RoboDK station: Enrega_Final.rdk

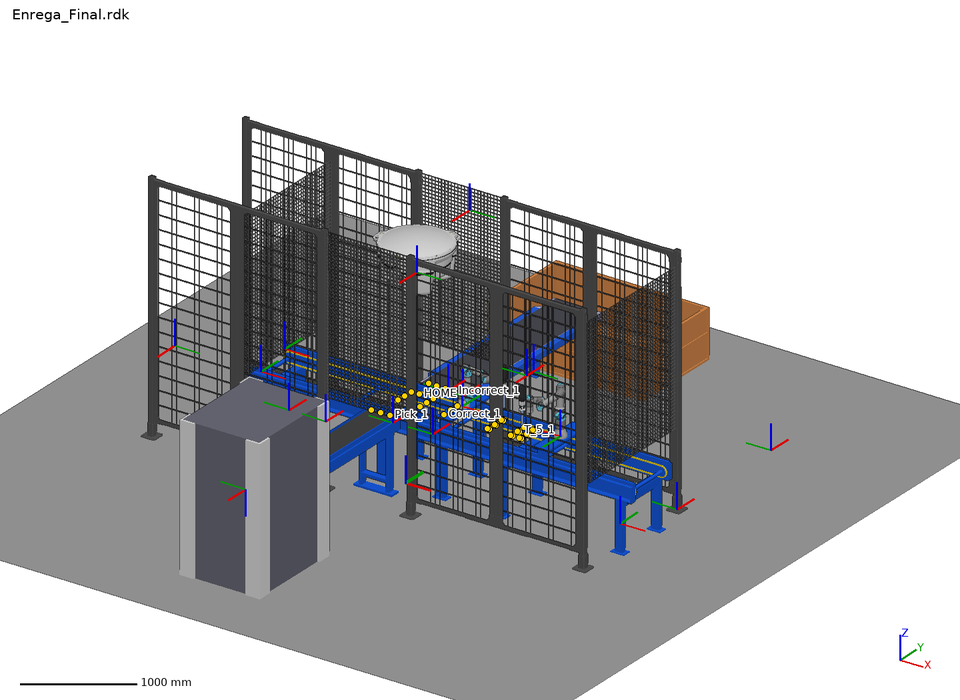
[picture v0: the station drawn from its stored meshes, robots at their saved joint values, targets as dots, program paths as lines]
Station Enrega_Final2 (saved by RoboDK 5.9.4). Poses are relative to the parent item; angles as X-Y-Z fixed-axis rotations.
Station parameters (name, value as stored): conv_pos, 0, groups_created, 0, stop, 0, group_counter_incorrectos, 0, conv_pos_exit, 0, groups_to_process, 0, serigrafia, 0, serigrafia1, 0, cinta_salida, 0, cinta_entrada, 0, salida_group_id, 0, salida_groups_on_belt, 0, salida_first_group_id, 0, main_conv_pos, 0, main_group_id, 0, main_groups_on_belt, 0, main_first_group_id, 0, cinta_central, 0, correct_group_id, 0, correct_groups_on_belt, 0, correct_first_group_id, 0, led_salida, 1, salir, 0
  - frame World at (0, 0, 0) mm
    - object Floor at (0, 0, 0) mm, size 7200 x 7200 x 0 mm, geometry from Floor.sld
    - frame MainConveyor Base at (-1580, 450, 650) mm
      - robot MainConveyor: 1 axes
          modified DH rows (alpha deg, a mm, theta deg, d mm): 0, 0, 0, 0 linear
          base shift (0, 0, 0) mm, rotated rx 0 ry 90 rz 0 deg
          joint limits [-200000] to [200000]; home [0]; saved at [0]
        - frame MainConveyorRef at (-800, -492, 0) mm, rotated rx 0 ry 0 rz -90 deg
      - frame MainConveyorRef_Init at (90, -480, 0) mm
    - frame UR3eBase1 at (1470, 200, 770) mm, rotated rx 0 ry 0 rz 180 deg
      - robot UR3e_1 (model UR3e): 6 axes, payload 3 kg, reach 500 mm, repeatability 0.03 mm, weight 11 kg
          modified DH rows (alpha deg, a mm, theta deg, d mm): 0, 0, 0, 151.9; 90, 0, 180, 0; 0, 243.55, 0, 0; 0, 213.2, 0, 131.05; -90, 0, 0, 85.35; 90, 0, 180, 92.1
          joint limits [-360, -360, -360, -360, -360, -360] to [360, 360, 360, 360, 360, 360]; home [0, -90, -90, 0, 90, 0]; saved at [38.708, -87.691, -123.564, -58.745, 90, 38.708]
        - tool Laser1, TCP at (0, -75, 221.24) mm, rotated rx 0 ry 0 rz 90 deg, size 63 x 128.2 x 432.2 mm
      - target T_5_1 (Cartesian target) at (453.12, -41.05, -88.71) mm, rotated rx -180 ry 0 rz -180 deg; joints [13.959, -117.749, -104.305, -47.946, 90, 13.959] of UR3e_1
      - target T_5_2 (Cartesian target) at (453.12, -31.05, -88.71) mm, rotated rx -180 ry 0 rz -180 deg; joints [15.513, -117.567, -104.617, -47.816, 90, 15.513] of UR3e_1
      - target T_5_3 (Cartesian target) at (453.12, -21.05, -88.71) mm, rotated rx -180 ry 0 rz -180 deg; joints [17.059, -117.435, -104.843, -47.722, 90, 17.059] of UR3e_1
      - target T_5_4 (Cartesian target) at (443.12, -21.05, -88.71) mm, rotated rx -180 ry 0 rz -180 deg; joints [17.546, -115.52, -108.09, -46.39, 90, 17.546] of UR3e_1
      - target T_5_5 (Cartesian target) at (463.12, -21.05, -88.71) mm, rotated rx -180 ry 0 rz -180 deg; joints [16.599, -119.355, -101.528, -49.117, 90, 16.599] of UR3e_1
      - target T_6_1 (Cartesian target) at (453.12, -141.05, -88.71) mm, rotated rx -180 ry 0 rz -180 deg; joints [-1.508, -122.242, -96.445, -51.314, 90, -1.508] of UR3e_1
      - target T_6_2 (Cartesian target) at (453.12, -131.05, -88.71) mm, rotated rx -180 ry 0 rz -180 deg; joints [0, -121.581, -97.617, -50.801, 90, 0] of UR3e_1
      - target T_6_3 (Cartesian target) at (453.12, -121.05, -88.71) mm, rotated rx -180 ry 0 rz -180 deg; joints [1.522, -120.967, -98.704, -50.329, 90, 1.522] of UR3e_1
      - target T_6_4 (Cartesian target) at (443.12, -121.05, -88.71) mm, rotated rx -180 ry 0 rz -180 deg; joints [1.564, -119.128, -101.923, -48.949, 90, 1.564] of UR3e_1
      - target T_6_5 (Cartesian target) at (463.12, -121.05, -88.71) mm, rotated rx -180 ry 0 rz -180 deg; joints [1.482, -122.826, -95.401, -51.773, 90, 1.482] of UR3e_1
      - target T_7_1 (Cartesian target) at (358.12, -136.05, -88.71) mm, rotated rx -180 ry 0 rz -180 deg; joints [-1.008, -104.831, -124.911, -40.258, 90, -1.008] of UR3e_1
      - target T_7_2 (Cartesian target) at (358.12, -126.05, -88.71) mm, rotated rx -180 ry 0 rz -180 deg; joints [1.016, -103.97, -126.152, -39.878, 90, 1.016] of UR3e_1
      - target T_7_3 (Cartesian target) at (358.12, -116.05, -88.71) mm, rotated rx -180 ry 0 rz -180 deg; joints [3.071, -103.155, -127.308, -39.536, 90, 3.071] of UR3e_1
      - target T_7_4 (Cartesian target) at (348.12, -116.05, -88.71) mm, rotated rx -180 ry 0 rz -180 deg; joints [3.186, -101.205, -130.002, -38.792, 90, 3.186] of UR3e_1
      - target T_7_5 (Cartesian target) at (368.12, -116.05, -88.71) mm, rotated rx -180 ry 0 rz -180 deg; joints [2.964, -105.064, -124.571, -40.364, 90, 2.964] of UR3e_1
      - target T_8_1 (Cartesian target) at (358.12, -41.05, -88.71) mm, rotated rx -180 ry 0 rz -180 deg; joints [19.014, -98.871, -133.084, -38.044, 90, 19.014] of UR3e_1
      - target T_8_2 (Cartesian target) at (358.12, -31.05, -88.71) mm, rotated rx -180 ry 0 rz -180 deg; joints [21.136, -98.589, -133.447, -37.965, 90, 21.136] of UR3e_1
      - target T_8_3 (Cartesian target) at (358.12, -21.05, -88.71) mm, rotated rx -180 ry 0 rz -180 deg; joints [23.239, -98.383, -133.709, -37.908, 90, 23.239] of UR3e_1
      - target T_8_4 (Cartesian target) at (348.12, -21.05, -88.71) mm, rotated rx -180 ry 0 rz -180 deg; joints [24.174, -96.082, -136.551, -37.367, 90, 24.174] of UR3e_1
      - target T_8_5 (Cartesian target) at (368.12, -21.05, -88.71) mm, rotated rx -180 ry 0 rz -180 deg; joints [22.376, -100.585, -130.837, -38.578, 90, 22.376] of UR3e_1
      - target T_9_1 (Cartesian target) at (358.12, 58.95, -88.71) mm, rotated rx -180 ry 0 rz -180 deg; joints [38.708, -99.562, -132.189, -38.249, 90, 38.708] of UR3e_1
      - target T_9_2 (Cartesian target) at (358.12, 68.95, -88.71) mm, rotated rx -180 ry 0 rz -180 deg; joints [40.414, -100.046, -131.554, -38.401, 90, 40.414] of UR3e_1
      - target T_9_3 (Cartesian target) at (358.12, 78.95, -88.71) mm, rotated rx -180 ry 0 rz -180 deg; joints [42.06, -100.595, -130.823, -38.581, 90, 42.06] of UR3e_1
      - target T_9_4 (Cartesian target) at (348.12, 78.95, -88.71) mm, rotated rx -180 ry 0 rz -180 deg; joints [43.571, -98.473, -133.594, -37.933, 90, 43.571] of UR3e_1
      - target T_9_5 (Cartesian target) at (368.12, 78.95, -88.71) mm, rotated rx -180 ry 0 rz -180 deg; joints [40.65, -102.65, -128.016, -39.334, 90, 40.65] of UR3e_1
    - frame UR3eBase2 at (450, 200, 770) mm
      - robot UR3e_2 (model UR3e): 6 axes, payload 3 kg, reach 500 mm, repeatability 0.03 mm, weight 11 kg
          modified DH rows (alpha deg, a mm, theta deg, d mm): 0, 0, 0, 151.9; 90, 0, 180, 0; 0, 243.55, 0, 0; 0, 213.2, 0, 131.05; -90, 0, 0, 85.35; 90, 0, 180, 92.1
          joint limits [-360, -360, -360, -360, -360, -360] to [360, 360, 360, 360, 360, 360]; home [0, -90, -90, 0, 90, 0]; saved at [54.922, -88.509, -122.462, -59.029, 90, 54.922]
        - tool Laser2, TCP at (0, -75, 221.24) mm, rotated rx 0 ry 0 rz 90 deg, size 63 x 128.2 x 432.2 mm
      - target T_3_1 (Cartesian target) at (332.71, -66.05, -87.69) mm, rotated rx -180 ry 0 rz -180 deg; joints [15.136, -93.886, -138.655, -37.459, 90, 15.136] of UR3e_2
      - target T_3_2 (Cartesian target) at (332.71, -76.05, -87.69) mm, rotated rx -180 ry 0 rz -180 deg; joints [12.75, -94.543, -137.908, -37.549, 90, 12.75] of UR3e_2
      - target T_3_3 (Cartesian target) at (332.71, -86.05, -87.69) mm, rotated rx -180 ry 0 rz -180 deg; joints [10.374, -95.271, -137.063, -37.666, 90, 10.374] of UR3e_2
      - target T_3_4 (Cartesian target) at (342.71, -86.05, -87.69) mm, rotated rx -180 ry 0 rz -180 deg; joints [9.959, -97.505, -134.367, -38.128, 90, 9.959] of UR3e_2
      - target T_3_5 (Cartesian target) at (322.71, -86.05, -87.69) mm, rotated rx -180 ry 0 rz -180 deg; joints [10.827, -92.927, -139.721, -37.351, 90, 10.827] of UR3e_2
      - target T_2_1 (Cartesian target) at (332.71, 33.95, -87.69) mm, rotated rx -180 ry 0 rz -180 deg; joints [37.78, -92.338, -140.361, -37.3, 90, 37.78] of UR3e_2
      - target T_2_2 (Cartesian target) at (332.71, 23.95, -87.69) mm, rotated rx -180 ry 0 rz -180 deg; joints [35.729, -92.048, -140.672, -37.279, 90, 35.729] of UR3e_2
      - target T_2_3 (Cartesian target) at (332.71, 13.95, -87.69) mm, rotated rx -180 ry 0 rz -180 deg; joints [33.614, -91.857, -140.876, -37.267, 90, 33.614] of UR3e_2
      - target T_2_4 (Cartesian target) at (342.71, 13.95, -87.69) mm, rotated rx -180 ry 0 rz -180 deg; joints [32.248, -94.39, -138.084, -37.527, 90, 32.248] of UR3e_2
      - target T_2_5 (Cartesian target) at (322.71, 13.95, -87.69) mm, rotated rx -180 ry 0 rz -180 deg; joints [35.108, -89.141, -143.636, -37.223, 90, 35.108] of UR3e_2
      - target T_1_1 (Cartesian target) at (332.71, 138.95, -87.69) mm, rotated rx -180 ry 0 rz -180 deg; joints [54.922, -100.1, -131.044, -38.857, 90, 54.922] of UR3e_2
      - target T_1_2 (Cartesian target) at (332.71, 128.95, -87.69) mm, rotated rx -180 ry 0 rz -180 deg; joints [53.632, -99.082, -132.372, -38.547, 90, 53.632] of UR3e_2
      - target T_1_3 (Cartesian target) at (332.71, 118.95, -87.69) mm, rotated rx -180 ry 0 rz -180 deg; joints [52.274, -98.107, -133.614, -38.279, 90, 52.274] of UR3e_2
      - target T_1_4 (Cartesian target) at (342.71, 118.95, -87.69) mm, rotated rx -180 ry 0 rz -180 deg; joints [50.531, -100.136, -130.996, -38.868, 90, 50.531] of UR3e_2
      - target T_1_5 (Cartesian target) at (322.71, 118.95, -87.69) mm, rotated rx -180 ry 0 rz -180 deg; joints [54.134, -96.01, -136.188, -37.801, 90, 54.134] of UR3e_2
      - target T_4_1 (Cartesian target) at (567.71, -61.05, -87.69) mm, rotated rx -180 ry 0 rz -180 deg; joints [8.242, -142.641, -57.678, -69.681, 90, 8.242] of UR3e_2
      - target T_4_2 (Cartesian target) at (567.71, -71.05, -87.69) mm, rotated rx -180 ry 0 rz -180 deg; joints [7.058, -143.003, -56.966, -70.031, 90, 7.058] of UR3e_2
      - target T_4_3 (Cartesian target) at (567.71, -81.05, -87.69) mm, rotated rx -180 ry 0 rz -180 deg; joints [5.874, -143.422, -56.139, -70.439, 90, 5.874] of UR3e_2
      - target T_4_4 (Cartesian target) at (577.71, -81.05, -87.69) mm, rotated rx -180 ry 0 rz -180 deg; joints [5.755, -146.272, -50.488, -73.24, 90, 5.755] of UR3e_2
      - target T_4_5 (Cartesian target) at (557.71, -81.05, -87.69) mm, rotated rx -180 ry 0 rz -180 deg; joints [5.998, -140.79, -61.31, -67.9, 90, 5.998] of UR3e_2
    - frame StickConveyor Base at (0, -190, 640) mm, rotated rx 0 ry 0 rz 90 deg
      - robot StickConveyorDoor: 1 axes
          modified DH rows (alpha deg, a mm, theta deg, d mm): 0, 0, 0, 0 linear
          joint limits [0] to [80]; home [0]; saved at [10]
        - frame GreenLedref1 at (450, 335, 1075) mm, rotated rx 0 ry 90 rz 0 deg
          - object Light (Green)1 at (0, 0, 0) mm, size 56 x 56 x 103.8 mm, geometry from Light-Green.sld
        - frame RedLedref1 at (450, 335, 1075) mm, rotated rx 0 ry 90 rz 0 deg
          - object Light (Red)1 at (0, 0, 0) mm, size 56 x 56 x 103.8 mm, geometry from Light-Red.sld
        - frame GreenLedref2 at (450, -50, 1075) mm, rotated rx 0 ry 90 rz 0 deg
          - object Light (Green)2 at (0, 0, 0) mm, size 56 x 56 x 103.8 mm, geometry from Light-Green.sld
        - frame RedLedref2 at (450, -50, 1075) mm, rotated rx 0 ry 90 rz 0 deg
          - object Light (Red)2 at (0, 0, 0) mm, size 56 x 56 x 103.8 mm, geometry from Light-Red.sld
      - robot StickConveyor: 1 axes
          modified DH rows (alpha deg, a mm, theta deg, d mm): 0, 0, 0, 0 linear
          base shift (0, 0, 0) mm, rotated rx 0 ry 90 rz 0 deg
          joint limits [-200000] to [200000]; home [0]; saved at [0]
        - frame StickConveyorRef at (-1965, 162.5, 110) mm, rotated rx -180 ry 0 rz 180 deg
      - object Camara at (-1460, -150, 480) mm, rotated rx 0 ry 90 rz 0 deg, size 101 x 460.9 x 328.2 mm, geometry from Camara.stl
        - object OpenCV OAK-D Camera at (75, 300, 450) mm, rotated rx 90 ry 0 rz 90 deg, size 110 x 54.5 x 33 mm, geometry from OpenCV-OAK-D-Camera (1).sld
    - frame DelteConveyor Base at (-350, 2400, 0) mm, rotated rx 0 ry 0 rz -90 deg
      - object Conveyor_legs_salida at (0, 0, 0) mm, size 1624 x 606 x 631 mm, geometry from Conveyor_legs_salida.stl
      - frame Conveyor Out Base at (1800, 522.5, 635) mm, rotated rx 0 ry 0 rz 180 deg
        - robot Conveyor Out: 1 axes
            modified DH rows (alpha deg, a mm, theta deg, d mm): 0, 0, 0, 0 linear
            base shift (0, 0, 0) mm, rotated rx 0 ry 90 rz 0 deg
            joint limits [-500000] to [500000]; home [0]; saved at [0]
          - frame DeleteStickConveyorRef at (0, 152.5, 0) mm
      - object Container at (-50, -500, 0) mm, size 1000 x 1600 x 500 mm, geometry from Container.stl
    - frame DeltaRobot_Base at (400, 380, 2550) mm, rotated rx 0 ry 0 rz -90 deg
      - frame ABB IRB 360-1/800 4D Base at (160, -440, -650) mm
        - robot ABB IRB 360-1/800 4D: 4 axes, payload 1 kg, reach 400 mm, repeatability 0.04 mm, weight 120 kg
            joint limits [-42, -42, -42, -36000] to [99.5, 99.5, 99.5, 36000]; home [0, 0, 0, 0]; saved at [4.542, 3.41, -0.23, 90]
          - tool RobotiQ EPick Vacuum Gripper (1 Cup), TCP at (0, 0, 130) mm, size 75 x 83 x 136.1 mm
        - target HOME (Cartesian target) at (-14.81, 15.75, -1155.85) mm, rotated rx 180 ry 0 rz -90 deg; joints [4.542, 3.41, -0.23, 90, 90, 0] of ABB IRB 360-1/800 4D
        - target Pick_1 (Cartesian target) at (415.27, 9.37, -1193.06) mm, rotated rx 180 ry 0 rz 0 deg; joints [-13.094, 63.364, 61.798, 0] of ABB IRB 360-1/800 4D
        - target Pick_2 (Cartesian target) at (415.27, -85.63, -1193.06) mm, rotated rx 180 ry 0 rz 0 deg; joints [-11.969, 56.404, 70.688, 0] of ABB IRB 360-1/800 4D
        - target Pick_3 (Cartesian target) at (415.27, -185.63, -1193.06) mm, rotated rx 180 ry 0 rz 0 deg; joints [-7.726, 51.888, 82.789, 0] of ABB IRB 360-1/800 4D
        - target Correct_1 (Cartesian target) at (90.27, 344.37, -1218.06) mm, rotated rx 180 ry 0 rz -90 deg; joints [26.179, 71.103, 5.738, 90] of ABB IRB 360-1/800 4D
        - target Correct_2 (Cartesian target) at (90.27, 94.37, -1218.06) mm, rotated rx 180 ry 0 rz -90 deg; joints [8.409, 33.6, 14.921, 90] of ABB IRB 360-1/800 4D
        - target Correct_3 (Cartesian target) at (90.27, -135.63, -1218.06) mm, rotated rx 180 ry 0 rz -90 deg; joints [9.908, 12.097, 38.803, 90] of ABB IRB 360-1/800 4D
        - target Correct_4 (Cartesian target) at (-9.73, 344.37, -1218.06) mm, rotated rx 180 ry 0 rz -90 deg; joints [36.874, 65.68, -1.742, 90] of ABB IRB 360-1/800 4D
        - target Correct_7 (Cartesian target) at (-109.73, 344.37, -1218.06) mm, rotated rx 180 ry 0 rz -90 deg; joints [50.145, 63.347, -5.955, 90] of ABB IRB 360-1/800 4D
        - target Correct_5 (Cartesian target) at (-9.73, 94.37, -1218.06) mm, rotated rx 180 ry 0 rz -90 deg; joints [19.165, 26.881, 7.588, 90] of ABB IRB 360-1/800 4D
        - target Correct_6 (Cartesian target) at (-9.73, -135.63, -1218.06) mm, rotated rx 180 ry 0 rz -90 deg; joints [20.646, 4.702, 32.281, 90] of ABB IRB 360-1/800 4D
        - target Correct_8 (Cartesian target) at (-109.73, 94.37, -1218.06) mm, rotated rx 180 ry 0 rz -90 deg; joints [32.347, 23.028, 3.333, 90] of ABB IRB 360-1/800 4D
        - target Correct_9 (Cartesian target) at (-109.73, -135.63, -1218.06) mm, rotated rx 180 ry 0 rz -90 deg; joints [33.81, 0.428, 28.596, 90] of ABB IRB 360-1/800 4D
        - target Incorrect_2 (Cartesian target) at (-394.73, 19.37, -1258.06) mm, rotated rx -180 ry 0 rz -180 deg; joints [88.789, 29.348, 25.106, 180] of ABB IRB 360-1/800 4D
        - target Incorrect_3 (Cartesian target) at (-394.73, -70.63, -1258.06) mm, rotated rx -180 ry 0 rz -180 deg; joints [89.794, 20.28, 35.776, 180] of ABB IRB 360-1/800 4D
        - target Incorrect_4 (Cartesian target) at (-394.73, -150.63, -1258.06) mm, rotated rx -180 ry 0 rz -180 deg; joints [93.919, 14.486, 47.855, 180] of ABB IRB 360-1/800 4D
        - target Incorrect_1 (Cartesian target) at (-394.73, 109.37, -1258.06) mm, rotated rx -180 ry 0 rz -180 deg; joints [91.364, 41.292, 17.211, 180] of ABB IRB 360-1/800 4D
    - frame Celda1 at (-350, 900, 0) mm, rotated rx 0 ry 0 rz 90 deg
      - object celda at (0, 150, 0) mm, size 146 x 1946 x 2470 mm, geometry from celda.stl
        - object mallacelda at (0, 0, 0) mm, size 1 x 756.4 x 2225.7 mm, geometry from mallacelda.stl
        - object mallacelda at (0, 900, 0) mm, size 1 x 756.4 x 2225.7 mm, geometry from mallacelda.stl
    - frame Celda2 at (2200, 900, 0) mm, rotated rx 0 ry 0 rz 90 deg
      - object celda at (0, 0, 0) mm, size 146 x 1946 x 2470 mm, geometry from celda.stl
        - object mallacelda at (0, 0, 0) mm, size 1 x 756.4 x 2225.7 mm, geometry from mallacelda.stl
        - object mallacelda at (0, 900, 0) mm, size 1 x 756.4 x 2225.7 mm, geometry from mallacelda.stl
        - object malla at (-1410, 2160, 1500) mm, rotated rx 0 ry 90 rz 0 deg, size 889.3 x 889.3 x 8.9 mm, geometry from malla.stl
        - object malla at (-1410, 2160, 2185) mm, rotated rx 0 ry 90 rz 0 deg, size 889.3 x 889.3 x 8.9 mm, geometry from malla.stl
        - object malla at (-850, 3590, 1400) mm, rotated rx 0 ry 90 rz 90 deg, size 889.3 x 889.3 x 8.9 mm, geometry from malla.stl
        - object malla at (-370, 3590, 1400) mm, rotated rx 0 ry 90 rz 90 deg, size 889.3 x 889.3 x 8.9 mm, geometry from malla.stl
        - object malla at (-850, 3590, 2050) mm, rotated rx 0 ry 90 rz 90 deg, size 889.3 x 889.3 x 8.9 mm, geometry from malla.stl
        - object malla at (-370, 3590, 2050) mm, rotated rx 0 ry 90 rz 90 deg, size 889.3 x 889.3 x 8.9 mm, geometry from malla.stl
    - frame Celda3 at (2200, 2300, 0) mm, rotated rx 0 ry 0 rz 90 deg
      - object celda at (0, 0, 0) mm, size 146 x 1946 x 2470 mm, geometry from celda.stl
        - object mallacelda at (0, 0, 0) mm, size 1 x 756.4 x 2225.7 mm, geometry from mallacelda.stl
        - object mallacelda at (0, 900, 0) mm, size 1 x 756.4 x 2225.7 mm, geometry from mallacelda.stl
        - object malla at (-1410, 2160, 1500) mm, rotated rx 0 ry 90 rz 0 deg, size 889.3 x 889.3 x 8.9 mm, geometry from malla.stl
        - object malla at (-1410, 2160, 2185) mm, rotated rx 0 ry 90 rz 0 deg, size 889.3 x 889.3 x 8.9 mm, geometry from malla.stl
    - frame Celda4 at (-350, 2300, 0) mm, rotated rx 0 ry 0 rz 90 deg
      - object celda at (0, 150, 0) mm, size 146 x 1946 x 2470 mm, geometry from celda.stl
        - object mallacelda at (0, 0, 0) mm, size 1 x 756.4 x 2225.7 mm, geometry from mallacelda.stl
        - object mallacelda at (0, 900, 0) mm, size 1 x 756.4 x 2225.7 mm, geometry from mallacelda.stl
        - object malla at (-2250, -2710, 1400) mm, rotated rx 0 ry 90 rz 90 deg, size 889.3 x 889.3 x 8.9 mm, geometry from malla.stl
        - object malla at (-1770, -2710, 1400) mm, rotated rx 0 ry 90 rz 90 deg, size 889.3 x 889.3 x 8.9 mm, geometry from malla.stl
        - object malla at (-2250, -2710, 2050) mm, rotated rx 0 ry 90 rz 90 deg, size 889.3 x 889.3 x 8.9 mm, geometry from malla.stl
        - object malla at (-1770, -2710, 2050) mm, rotated rx 0 ry 90 rz 90 deg, size 889.3 x 889.3 x 8.9 mm, geometry from malla.stl
        - object BotonStop at (-1310, 80, 1500) mm, rotated rx 0 ry 0 rz 180 deg, size 128.4 x 103.1 x 104 mm, geometry from Emergency_Stop.obj
    - frame Plantilla3 at (1900, 483.3, -50) mm
      - object AssemblyRack at (0, 0, 0) mm, rotated rx 0 ry 0 rz 90 deg, size 485 x 853 x 40 mm, geometry from AssemblyRack.step
        - object Plantilla3 at (-100, 535, 45) mm, rotated rx 180 ry 0 rz 90 deg, size 817.7 x 452.4 x 35.3 mm, geometry from Plantilla3.stl
  - folder StickConveyor
    - Python program StickConveyorMove (listed below)
    - Python program ResetStickConveyor (listed below)
    - Python program StickConveyorDeleteMove (listed below)
    - Python program ResetStickConveyorDeleteMove (listed below)
  - frame StickFrameCorrecto at (0, 0, -10) mm
    - object StickCorrecto at (-50, 35, -50) mm, size 197.9 x 35.6 x 6.3 mm, geometry from palillod.stl
  - frame StickFrameIncorrecto at (0, 0, -10) mm
    - object StickIncorrecto at (-50, 35, -50) mm, size 197.9 x 35.6 x 6.3 mm, geometry from palillod.stl
  - folder ScriptDelta
    - Python program Delta (listed below)
    - Python program ResetDelta (listed below)
    - Python program ResetPalillo (listed below)
  - folder ScriptSerigrafia
    - Python program SerigrafiaUR3e2 (listed below)
    - Python program SerigrafiaUR3e1 (listed below)
    - Python program WeldOn (listed below)
    - Python program ResetSoldar (listed below)
  - folder BasedeDatos
    - Python program ConexionBasedeDatos (listed below)
  - folder Mqtt
    - Python program MqttListener (listed below)
    - Python program RobotController (listed below)
  - folder CintaCentral
    - Python program MainConveyor (listed below)
    - Python program ResetMainConveyor (listed below)
  - folder ResetGeneral
    - Python program ResetGeneral (listed below)
    - Python program PararProgramas (listed below)
  - folder BotonStop
    - Python program StopBoton (listed below)
  - folder Main
    - Python program ProgramaPrincipal (listed below)

--- Python program StickConveyorMove ---
import sys
sys.path.append(r"C:\Users\Fran\Downloads\ProyectoPrueba")
import MqttListener as mqtt_listener
from ConexionBasedeDatos import crear_proceso_y_palillo
from robodk import robolink
from robodk.robomath import transl
from robodk.robodialogs import mbox
import random
import time

RDK = robolink.Robolink()

FRAME = RDK.Item('StickConveyorRef', robolink.ITEM_TYPE_FRAME)
stick_ok = RDK.Item('StickCorrecto', robolink.ITEM_TYPE_OBJECT)
stick_no = RDK.Item('StickIncorrecto', robolink.ITEM_TYPE_OBJECT)
led_verde = RDK.Item('Light (Green)2', robolink.ITEM_TYPE_OBJECT)
led_rojo = RDK.Item('Light (Red)2', robolink.ITEM_TYPE_OBJECT)

mqtt_listener.conectar_mqtt()
mqtt_listener.iniciar_loop_mqtt()
time.sleep(1)

nombre = mbox("Introduce el nombre:", entry="")

mqtt_listener.publicar_lcd(nombre)

STEP_GROUP = 400
OFFSET_Y = 100
MAX_GROUPS = 5

def esperar_stop():
        while int(RDK.getParam("stop") or 0) == 1:
                time.sleep(0.1)


def led_verde_on():
        global ultimo_led_entrada

        led_verde.setVisible(True)
        led_rojo.setVisible(False)
        if ultimo_led_entrada != 1:
                mqtt_listener.encender_led()
                print("MQTT entrada: ENCENDER_LED")
                ultimo_led_entrada = 1

        RDK.Update()

def led_rojo_on():
        global ultimo_led_entrada

        led_verde.setVisible(False)
        led_rojo.setVisible(True)
        if ultimo_led_entrada != 0:
                mqtt_listener.apagar_led()
                print("MQTT entrada: APAGAR_LED")
                ultimo_led_entrada = 0
        RDK.Update()

def move_cinta(step=STEP_GROUP):
    mechanism = RDK.Item('StickConveyor', robolink.ITEM_TYPE_ROBOT)
    if mechanism.Valid():
        j = mechanism.Joints()
        current = j[0, 0]
        mechanism.setJoints([current + float(step)])

RDK.Render(True)

ultimo_led_salida = None
ultimo_led_entrada = None

conveyor_position = float(RDK.getParam('conv_pos') or 0)
fin_notificado = False

while int(RDK.getParam("salir") or 0) == 0:

    esperar_stop()

    groups_created = int(RDK.getParam('groups_created') or 0)
    groups_to_process = int(RDK.getParam('groups_to_process') or 0)

    led_salida_param = RDK.getParam('led_salida')

    if led_salida_param is None or led_salida_param == '':
            led_salida = 1
    else:
            led_salida = int(led_salida_param)

    if led_salida != ultimo_led_salida:

            if led_salida == 1:
                mqtt_listener.encender_led_2()
                print("MQTT salida: ENCENDER_LED")
            else:
                mqtt_listener.apagar_led_2()
                print("MQTT salida: APAGAR_LED")

            ultimo_led_salida = led_salida

    pending = groups_created - groups_to_process

    if pending < MAX_GROUPS:

        fin_notificado = False

        group_id = groups_created

        print("Creando grupo", group_id)

        RDK.Render(False)

        for i in range(3):

            selected = random.choice([stick_ok, stick_ok, stick_ok, stick_ok, stick_no])

            selected.Copy()
            obj = RDK.Paste()

            if not obj.Valid():
                print("Paste falló")
                continue

            obj.setParent(FRAME)

            y_offset = (i - 1) * OFFSET_Y

            obj.setPose(transl(conveyor_position,y_offset,0))

            es_correcto = selected.Name() == stick_ok.Name()

            obj.setName(
                f"{'correcto' if es_correcto else 'incorrecto'}_{group_id}_{i}"
            )
            if es_correcto:
                    crear_proceso_y_palillo()

        conveyor_position += STEP_GROUP
        RDK.setParam('conv_pos', str(conveyor_position))

        RDK.Render(True)

        led_rojo_on()
        time.sleep(0.1)

        esperar_stop()

        RDK.setParam('cinta_entrada', 1)

        try:
            move_cinta()
            time.sleep(0.2)
        finally:
            RDK.setParam('cinta_entrada', 0)

        led_verde_on()

        groups_created += 1

        RDK.setParam('groups_created', groups_created)

        RDK.Render(True)
        RDK.Update()

        time.sleep(0.5)

    else:
            if not fin_notificado:
                    RDK.Render(True)
                    led_verde_on()
                    fin_notificado = True
            time.sleep(0.1)

--- Python program ResetStickConveyor ---
# Type help("robodk.robolink") or help("robodk.robomath") for more information
# Press F5 to run the script
# Documentation: https://robodk.com/doc/en/RoboDK-API.html
# Reference:     https://robodk.com/doc/en/PythonAPI/robodk.html
# Note: It is not required to keep a copy of this file, your Python script is saved with your RDK project

from robodk import robolink

RDK = robolink.Robolink()

MECHANISM_NAME = 'StickConveyor'

mechanism = RDK.Item(MECHANISM_NAME, robolink.ITEM_TYPE_ROBOT)

# =========================
# 1) reset parámetro
# =========================
RDK.setParam('conv_pos', 0)
RDK.setParam('groups_created', 0)
RDK.setParam('groups_to_process', 0)
RDK.setParam('cinta_entrada', 0)

# =========================
# 2) reset posición física del conveyor
# =========================
if mechanism.Valid():
    mechanism.setJoints([0])

print("Conveyor reseteado a posición inicial")

--- Python program StickConveyorDeleteMove ---
import sys
sys.path.insert(0, r"C:\Users\Fran\Downloads\ProyectoPrueba")
from robodk import robolink
from robodk.robomath import transl
import random
import time

RDK = robolink.Robolink()

FRAME = RDK.Item('DeleteStickConveyorRef', robolink.ITEM_TYPE_FRAME)
led_verde = RDK.Item('Light (Green)1', robolink.ITEM_TYPE_OBJECT)
led_rojo = RDK.Item('Light (Red)1', robolink.ITEM_TYPE_OBJECT)


time.sleep(1)

STEP_GROUP = 400
MAX_GROUPS = 4
MAX_GROUPS_SALIDA = 4

def esperar_stop():
        while int(RDK.getParam("stop") or 0) == 1:
                time.sleep(0.1)

def led_verde_on():
        led_verde.setVisible(True)
        led_rojo.setVisible(False)
        RDK.setParam('led_salida', 1)
        RDK.Update()

def led_rojo_on():
        led_verde.setVisible(False)
        led_rojo.setVisible(True)
        RDK.setParam('led_salida', 0)
        RDK.Update()


def move_cinta(step=STEP_GROUP):
    mechanism = RDK.Item('Conveyor Out', robolink.ITEM_TYPE_ROBOT)
    if mechanism.Valid():
        j = mechanism.Joints()
        current = j[0, 0]
        mechanism.setJoints([current + float(step)])

def borrar_grupo_salida(group_id):
        for i in range(4):
                obj = RDK.Item(f"salida_{group_id}_{i}")
                if obj.Valid():
                        obj.Delete()

RDK.Render(True)

led_verde_on()

while int(RDK.getParam("salir") or 0) == 0:

    esperar_stop()

    counter_stick = int(RDK.getParam('group_counter_incorrectos') or 0)

    print("group_counter_incorrectos =", counter_stick)

    if counter_stick  >= MAX_GROUPS:

        esperar_stop()

        led_rojo_on()
        RDK.setParam('cinta_salida', 1)

        try:
                move_cinta()
                time.sleep(0.2)
        finally:
                RDK.setParam('cinta_salida', 0)

        # REINICIAR CONTADOR
        counter_stick = int(RDK.getParam('group_counter_incorrectos') or 0)
        RDK.setParam('group_counter_incorrectos', max(0, counter_stick - 4))

        groups_on_belt = int(RDK.getParam('salida_groups_on_belt') or 0)
        first_group_id = int(RDK.getParam('salida_first_group_id') or 0)

        groups_on_belt +=1

        if groups_on_belt > MAX_GROUPS_SALIDA:
                borrar_grupo_salida(first_group_id)
                first_group_id += 1
                groups_on_belt -= 1
        RDK.setParam('salida_groups_on_belt', groups_on_belt)
        RDK.setParam('salida_first_group_id', first_group_id)

        led_verde_on()

    time.sleep(0.1)

--- Python program ResetStickConveyorDeleteMove ---
# Type help("robodk.robolink") or help("robodk.robomath") for more information
# Press F5 to run the script
# Documentation: https://robodk.com/doc/en/RoboDK-API.html
# Reference:     https://robodk.com/doc/en/PythonAPI/robodk.html
# Note: It is not required to keep a copy of this file, your Python script is saved with your RDK project

from robodk import robolink

RDK = robolink.Robolink()

MECHANISM_NAME = 'Conveyor Out'

mechanism = RDK.Item(MECHANISM_NAME, robolink.ITEM_TYPE_ROBOT)

# =========================
# 1) reset parámetro
# =========================
RDK.setParam('cinta_salida', 0)
RDK.setParam('group_counter_incorrectos', 0)
RDK.setParam('salida_group_id', 0)
RDK.setParam('salida_groups_on_belt', 0)
RDK.setParam('salida_first_group_id', 0)
RDK.setParam('led_salida', 1)

# =========================
# 2) reset posición física del conveyor
# =========================
if mechanism.Valid():
    mechanism.setJoints([0])

print("Conveyor reseteado a posición inicial")

--- Python program Delta ---
import sys
sys.path.append(r"C:\Users\Fran\Downloads\ProyectoPrueba")
from MainConveyor import avanzar_y_crear_bandeja, inicializar_bandejas, borrar_bandeja, MAX_BANDEJAS
from robodk import robolink
from robodk.robomath import transl
import time

RDK = robolink.Robolink()

robot = RDK.Item('ABB IRB 360-1/800 4D', robolink.ITEM_TYPE_ROBOT)
ref_salida_mal = RDK.Item('DeleteStickConveyorRef', robolink.ITEM_TYPE_FRAME)
ref_salida_bien = RDK.Item('MainConveyorRef', robolink.ITEM_TYPE_FRAME)
tool = RDK.Item('RobotiQ EPick Vacuum Gripper (1 Cup)')
home = RDK.Item('HOME', robolink.ITEM_TYPE_TARGET)

robot.setSpeed(800, 600)

Z_APPROACH = transl(0, 0, -75)


pick = []
for i in range(1, 4):
    t = RDK.Item(f'Pick_{i}', robolink.ITEM_TYPE_TARGET)
    if not t.Valid():
        print(f"ERROR: Pick_{i} no existe")
    pick.append(t)

correct = [RDK.Item(f'Correct_{i}') for i in range(1, 10)]

incorrect = [RDK.Item(f'Incorrect_{i}') for i in range(1, 5)]

# -------------------------
# INDICES
# -------------------------
correct_index = 0
incorrect_index = 0
processed_correct = 0

def esperar_stop():
    while int(RDK.getParam("stop") or 0) == 1:
        time.sleep(0.1)

inicializar_bandejas()

def esperar_cintas_paradas():
    while True:
        esperar_stop()

        cinta_entrada = int(RDK.getParam('cinta_entrada') or 0)
        cinta_salida = int(RDK.getParam('cinta_salida') or 0)
        cinta_central = int(RDK.getParam('cinta_central') or 0)

        if cinta_entrada == 0 and cinta_salida == 0 and cinta_central == 0:
            time.sleep(0.2)
            break

        time.sleep(0.1)


def borrar_grupo_correctos(group_id):
    for i in range(9):
        obj = RDK.Item(f"correct_out_{group_id}_{i}")
        if obj.Valid():
            print("Eliminando correcto:", obj.Name())
            obj.Delete()


def esperar_serigrafia_terminada():
    while True:
        esperar_stop()

        serigrafia1 = int(RDK.getParam('serigrafia1') or 0)
        serigrafia = int(RDK.getParam('serigrafia') or 0)

        if serigrafia1 == 0 and serigrafia == 0:
            break

        time.sleep(0.1)


# -------------------------
# HELPERS
# -------------------------
def pre(target):
    esperar_stop()
    esperar_cintas_paradas()
    robot.MoveJ(target.Pose() * Z_APPROACH)

def pre_place_incorrecto(target):
    esperar_stop()
    esperar_cintas_paradas()
    robot.MoveJ(target.Pose() * Z_APPROACH)

def go_place_incorrecto(target):
    esperar_stop()
    esperar_cintas_paradas()
    robot.MoveL(target.Pose())

def go(target):
    esperar_stop()
    esperar_cintas_paradas()
    robot.MoveL(target.Pose())


# -------------------------
# LOOP PRINCIPAL
# -------------------------
while int(RDK.getParam("salir") or 0) == 0:

    esperar_stop()

    groups_to_process = int(RDK.getParam('groups_to_process') or 0)
    groups_created = int(RDK.getParam('groups_created') or 0)
    correct_group_id = int(RDK.getParam('correct_group_id') or 0)

    esperar_cintas_paradas()

    if groups_to_process >= groups_created:
        time.sleep(0.1)
        continue

    group_id = groups_to_process

    all_items = RDK.ItemList()

    sticks = []

    for item in all_items:
        name = item.Name()

        if not name:
            continue

        parts = name.split("_")

        if len(parts) != 3:
            continue

        tipo, grupo, indice = parts

        if tipo not in ["correcto", "incorrecto"]:
            continue

        if not grupo.isdigit() or not indice.isdigit():
            continue

        if int(grupo) != group_id:
            continue

        sticks.append(item)

    if len(sticks) < 3:
        time.sleep(0.1)
        continue

    sticks.sort(key=lambda x: int(x.Name().split("_")[2]))



    # CICLO 3 PALILLOS
    for i in range(3):
        esperar_stop()

        esperar_cintas_paradas()

        stick = sticks[i]

        tipo = stick.Name().split("_")[0]

        esperar_stop()
        # PICK
        pre(pick[i])
        go(pick[i])

        tool.AttachClosest()

        pre(pick[i])

        if tipo == "correcto":
            pre(correct[correct_index])
            go(correct[correct_index])

            tool.DetachAll(ref_salida_bien)

            stick.setName(f"correct_out_{correct_group_id}_{correct_index}")

            pre(correct[correct_index])

            correct_index += 1
            processed_correct +=1

            if processed_correct >= 9:

                print("GRUPO DE 9 CORRECTOS COMPLETADO")

                esperar_stop()

                robot.MoveJ(home)
                time.sleep(0.3)

                esperar_serigrafia_terminada()

                esperar_stop()

                correct_groups_on_belt = int(RDK.getParam('correct_groups_on_belt') or 0)
                correct_first_group_id = int(RDK.getParam('correct_first_group_id') or 0)
                groups_on_belt = int(RDK.getParam('main_groups_on_belt') or 0)
                first_group_id = int(RDK.getParam('main_first_group_id') or 0)

                if correct_groups_on_belt >= 2:

                    borrar_grupo_correctos(correct_first_group_id)

                    correct_first_group_id += 1
                    correct_groups_on_belt -= 1

                if groups_on_belt >= MAX_BANDEJAS:
                    borrar_bandeja(first_group_id)
                    first_group_id += 1
                    groups_on_belt -= 1

                RDK.setParam('main_groups_on_belt', groups_on_belt)
                RDK.setParam('main_first_group_id', first_group_id)

                avanzar_y_crear_bandeja()

                correct_groups_on_belt += 1

                RDK.setParam('correct_groups_on_belt', correct_groups_on_belt)
                RDK.setParam('correct_first_group_id', correct_first_group_id)

                correct_group_id += 1
                RDK.setParam('correct_group_id', correct_group_id)

                RDK.setParam("serigrafia", 1)
                RDK.setParam("serigrafia1", 1)

                processed_correct = 0
                correct_index = 0

                print("SERIGRAFÍA")

        elif tipo == "incorrecto":
            esperar_stop()

            robot.MoveJ(home)
            pre_place_incorrecto(incorrect[incorrect_index])
            go_place_incorrecto(incorrect[incorrect_index])

            tool.DetachAll(ref_salida_mal)

            salida_group_id = int(RDK.getParam('salida_group_id') or 0)
            stick.setName(f"salida_{salida_group_id}_{incorrect_index}")
            pre_place_incorrecto(incorrect[incorrect_index])
            esperar_stop()
            robot.MoveJ(home)

            incorrect_index += 1


            c = int(RDK.getParam('group_counter_incorrectos') or 0)
            c += 1
            RDK.setParam('group_counter_incorrectos', c)

            if incorrect_index >= 4:

                incorrect_index = 0
                salida_group_id += 1
                RDK.setParam('salida_group_id', salida_group_id)

    # -------------------------
    # FIN DE GRUPO
    # -------------------------
    groups_to_process += 1
    RDK.setParam('groups_to_process', groups_to_process)

    time.sleep(0.1)

--- Python program ResetDelta ---
from robodk import robolink
from robodk.robomath import transl
import time

RDK = robolink.Robolink()

robot = RDK.Item('ABB IRB 360-1/800 4D', robolink.ITEM_TYPE_ROBOT)
home = RDK.Item('HOME', robolink.ITEM_TYPE_TARGET)

robot.setSpeed(800, 600)

robot.MoveJ(home)

--- Python program ResetPalillo ---
from robodk import robolink
import re

RDK = robolink.Robolink()

all_items = RDK.ItemList()

for item in all_items:

    name = item.Name()

    if not name:
        continue

    # correcto_0_1 / incorrecto_3_2
    patron_entrada = r'^(correcto|incorrecto)_\d+_\d+$'

    # salida_0_1
    patron_salida = r'^salida_\d+_\d+$'

    patron_correcto_salida = r'^correct_out_\d+_\d+$'

    if re.match(patron_entrada, name) or re.match(patron_salida, name) or re.match(patron_correcto_salida, name):

        print("Eliminando:", name)

        item.Delete()

print("Limpieza completada")

--- Python program SerigrafiaUR3e2 ---
from robodk import robolink, robomath
import time

RDK = robolink.Robolink()
RDK.setRunMode(robolink.RUNMODE_SIMULATE)
RDK.setSimulationSpeed(1)

robot = RDK.Item('UR3e_2')
tool = RDK.Item('Laser2')

if not robot.Valid():
    raise Exception("No existe el robot UR3e_2")

if not tool.Valid():
    raise Exception("No hay tool activa")

robot.setRounding(20)

Z_APPROACH = robomath.transl(0, 0, -60)

palillos = [
    (["T_1_1", "T_1_2", "T_1_3", "T_1_4", "T_1_5"]),
    (["T_2_1", "T_2_2", "T_2_3", "T_2_4", "T_2_5"]),
    (["T_3_1", "T_3_2", "T_3_3", "T_3_4", "T_3_5"]),
    (["T_4_1", "T_4_2", "T_4_3", "T_4_4", "T_4_5"])
]

def esperar_stop():
    while int(RDK.getParam("stop") or 0) == 1:
        time.sleep(0.1)


while int(RDK.getParam("salir") or 0) == 0:

    esperar_stop()

    # Esperar hasta que serigrafia sea 1
    if int(RDK.getParam("serigrafia") or 0) == 0:
        time.sleep(0.1)
        continue

    print("SERIGRAFIA ACTIVADA")

    for i, (target_names) in enumerate(palillos):

        esperar_stop()

        targets = [RDK.Item(name) for name in target_names]

        for t in targets:
            if not t.Valid():
                raise Exception("Falta target: " + t.Name())

        pre_inicio = targets[0].Pose() * Z_APPROACH
        pre_final = targets[-1].Pose() * Z_APPROACH

        robot.setSpeed(80, 40)

        esperar_stop()

        if i == 0:
            robot.MoveJ(pre_inicio)
        else:
            robot.setSpeed(60, 30)
            robot.MoveJ(pre_inicio)

        robot.setSpeed(30, 15)

        esperar_stop()

        robot.MoveL(targets[0])

        for t in targets[1:]:
            esperar_stop()
            robot.MoveL(t)

        esperar_stop()
        robot.MoveL(pre_final)

    inicio = RDK.Item('T_1_1')
    inicio1 = RDK.Item('T_3_5')

    preinicio = inicio.Pose() * Z_APPROACH
    preinicio1 = inicio1.Pose() * Z_APPROACH

    robot.setSpeed(60, 30)
    esperar_stop()
    robot.MoveJ(preinicio1)
    esperar_stop()
    robot.MoveJ(preinicio)

    RDK.setParam("serigrafia", 0)

    print("FIN SERIGRAFIA")

--- Python program SerigrafiaUR3e1 ---
from robodk import robolink, robomath
import time

RDK = robolink.Robolink()
RDK.setRunMode(robolink.RUNMODE_SIMULATE)
RDK.setSimulationSpeed(1)

robot = RDK.Item('UR3e_1')
tool = RDK.Item('Laser1')

if not robot.Valid():
    raise Exception("No existe el robot UR3e_1")

# Suavizado
robot.setRounding(20)

robot.setTool(tool)

# Offset de aproximación
Z_APPROACH = robomath.transl(0, 0, -60)

palillos = [
    (["T_9_1", "T_9_2", "T_9_3", "T_9_4", "T_9_5"]),
    (["T_8_1", "T_8_2", "T_8_3", "T_8_4", "T_8_5"]),
    (["T_7_1", "T_7_2", "T_7_3", "T_7_4", "T_7_5"]),
    (["T_6_1", "T_6_2", "T_6_3", "T_6_4", "T_6_5"]),
    (["T_5_1", "T_5_2", "T_5_3", "T_5_4", "T_5_5"]),
]

def esperar_stop():
    while int(RDK.getParam("stop") or 0) == 1:
        time.sleep(0.1)


while int(RDK.getParam("salir") or 0) == 0:

    esperar_stop()
    # Esperar activación
    if int(RDK.getParam("serigrafia1") or 0) == 0:
        time.sleep(0.1)
        continue

    print("SERIGRAFIA ACTIVADA")

    for i, (target_names) in enumerate(palillos):

        esperar_stop()

        targets = [RDK.Item(name) for name in target_names]

        for t in targets:
            if not t.Valid():
                raise Exception("Falta target: " + t.Name())

        pre_inicio = targets[0].Pose() * Z_APPROACH
        pre_final = targets[-1].Pose() * Z_APPROACH

        # -------------------------
        # MOVIMIENTO RÁPIDO
        # -------------------------
        robot.setSpeed(80, 40)

        esperar_stop()

        if i == 0:
            robot.MoveJ(pre_inicio)
        else:
            robot.setSpeed(60, 30)
            robot.MoveJ(pre_inicio)

        # -------------------------
        # MOVIMIENTO SUAVE
        # -------------------------
        robot.setSpeed(30, 15)

        esperar_stop()

        robot.MoveL(targets[0])

        RDK.RunProgram("WeldOn(ON)")

        for t in targets[1:]:
            esperar_stop()
            robot.MoveL(t)

        RDK.RunProgram("WeldOn(OFF)")

        esperar_stop()
        robot.MoveL(pre_final)

    # -------------------------
    # VOLVER A INICIO
    # -------------------------
    inicio = RDK.Item('T_9_1')
    preinicio = inicio.Pose() * Z_APPROACH

    if not inicio.Valid():
        raise Exception("No existe T_9_1")

    robot.setSpeed(60, 30)

    esperar_stop()

    robot.MoveJ(preinicio)

    # Reset del parámetro
    RDK.setParam("serigrafia1", 0)

    print("FIN SERIGRAFIA")

--- Python program WeldOn ---
# This macro allows simulating the material deposition of a weld gun
# By default, this macro will activate the trace once it is called.
# Run the macro ArcEnd to stop the trace.
#
# The macros ArcStart, ArcEnd and WeldOn, SpindleOn, all behave in a similar way, the only difference is the default behavior
# This behavior simmulates Fanuc Arc Welding and triggers appropriate output when using the customized post processor.
# Select ESC to clear the trace manually.
#
# It is possible to call WeldOn(ON) to simulate turning the material deposition ON or WeldOn(OFF) to stop simulating the gun
# Calling WeldOn(RESET) clears all displayed data.
# The macro will output spray gun statistics
#
# Optional:
#     This macro can manage multiple guns and multiple colors.
#     As an example, you can call this macro the following way:
#
# WeldOn(State, ToolName, Color)
#     State: [ON/OFF/RESET]
#     TorchName: The name of the tool. For example: Tool 1
#     Color: A named color or a hex color in the format: '#AARRGGBB'
#             Important: for full color definition you should provide Alpha channel first
#
# Examples:
#     WeldOn(ON)                 # Turn on the trace using the default color
#     WeldOn(OFF)                # Turn off the tool trace
#     WeldOn(ON, Tool 1, yellow) # Turn on the trace for tool 1 in yellow
#     WeldOn(ON, Tool 2, blue) # Turn on the trace for tool 2 in blue
#     WeldOn(OFF, Torch1)        # Turn off trace for Torch 1
#     WeldOn(ON, Torch1, #889900FF) # Turn on the trace for torch 2 in a violet color
#     WeldOn(ON, ,red)         # Turn on the trace for a generic torch in red color
#
# --------------------------------------------------------------
# This script shows how to create "spray" object in RoboDK that allows simulating particle deposition by using:
# RDK.Spray_Add(tool, object, options_command, volume, geometry)
#    tool: tool item (TCP) to use
#    object: object to project the particles
#    options_command (optional): string to specify options.
#    volume (optional): Matrix of parameters defining the volume of the spray gun
#    geometry (optional): Matrix of vertices defining the triangles.
#
# More information here:
# https://robodk.com/doc/en/PythonAPI/robodk.html#robodk.robolink.Robolink.Spray_Add
# https://robodk.com/doc/en/RoboDK-API.html
#
# The scripts ArcStart, ArcEnd and WeldOn and SpindleOn behave in a similar way, the only difference is the default behavior
# This behavior simmulates Fanuc Arc Welding and triggers appropriate output when using the customized post processor.
# Select ESC to clear the trace manually.
#
# Example scripts that use Spray_Add:
#     SpindleOn / SpindleOff    -> Turn trace On/Off
#     ArcOn / ArcOff            -> Turn trace On/Off
#     SprayOn / SprayOff        -> Simulate a spray given a workspace volume (for painting)
#     WeldOn / WeldOff          -> Support for multiple weld guns
#
#----------------------------------------------------------

# Constant variables for the first parameter:
ACTION_RESET = -1  # Same as: RESET (clear all traces)
ACTION_OFF = 0  # Same as: OFF (turn on)
ACTION_ON = 1  # Same as: ON (turn off)

# Define the default Action (ACTION_OFF to deactivate, ACTION_ON to activate, ACTION_RESET to clear any spray gun/trace)
# Setting it to None will display a message
Action = ACTION_ON

# Define the default color as a named color or as #AARRGGBB (Alpha, Red, Green Blue)
# COLOR = 'blue'
COLOR = 'red'  # AARRGGBB

# Use a specific tool as a spray gun
Tool_Name = None  # Use the active tool
#Tool_Name = 'Torch1'

# Use a specific object to project particles:
Object_Name = None  # Use the first object in the active reference frame
#Object_Name = 'Part'

# --------------------------------------------------
# Program start:
from robodk.robolink import *  # API to communicate with RoboDK
from robodk.robodialogs import *

RDK = Robolink()

# quit if we are not in simulation mode
if RDK.RunMode() != RUNMODE_SIMULATE:
    quit()

# Check command input (parameters passed in the call). This is the same as if we were doing a command line call passing parameters.
import sys
if len(sys.argv) > 1:
    Action_str = sys.argv[1].strip().upper()
    if 'ON' in Action_str:
        Action = ACTION_ON
    elif 'OFF' in Action_str:
        Action = ACTION_OFF
    elif 'RESET' in Action_str:
        Action = ACTION_RESET
    else:
        Action = int(Action_str)

    if len(sys.argv) > 2:
        Tool_Name = sys.argv[2].strip()
        if Tool_Name == '':
            Tool_Name = None

        if len(sys.argv) > 3:
            COLOR = sys.argv[3].lower().strip()

# Display summary
print("Applying action: " + str(Action))
print("Using tool: " + str(Tool_Name))
print("Using color: " + COLOR)

# Get any previously added spray gun simulations and display statistics (spray on the part vs spray falling out of the part)
info, data = RDK.Spray_GetStats()
n_sprays = data.size(1)
spray_id = -1
if n_sprays > 0 and Tool_Name is not None:
    spray_id = RDK.getParam(Tool_Name)
    if spray_id is None or Action == ACTION_ON or type(spray_id) == str or spray_id >= n_sprays:
        spray_id = -1

    print("Spray gun statistics:")
    print(info)
    print(data.tr())
    # # Diplay statistics
    # RDK.ShowMessage("Material used: %.1f%%<br>Material waisted: %.1f%%<br>Total particles: %.1f" % (data[1,0],data[2,0],data[3,0]), True)
    # # Clear previous spray
    # RDK.Spray_Clear()

# If the default Action is None, display a message to activate/deactivate the spray gun
if Action is None:
    print('Note: This macro can be called as ArcStart(1) or ArcStart(0) or ArcStart(-1)')
    entry = mbox('Turn gun ON or OFF', ('On', '1'), ('Off', '0'))
    if not entry:
        quit()
    Action = int(entry)

# Apply the desired action
if Action == ACTION_OFF:
    # Turn the gun off
    RDK.Spray_SetState(SPRAY_OFF, spray_id)

elif Action == ACTION_OFF:
    # Clear all spray simulations (same as pressing ESC key)
    RDK.Spray_Clear(spray_id)

elif Action == ACTION_ON:
    # Create a new spray gun object in RoboDK
    # by using RDK.Spray_Add(tool, object, options_command, volume, geometry)
    # tool: tool item (TCP) to use
    # object: object to project the particles
    # options_command (optional): string to specify options. Example:
    #     STEP=AxB: Defines the grid to be projected 1x1 means only one line of particle projection (for example, for welding)
    #     PARTICLE: Defines the shape and size of particle (sphere or particle), unless a specific geometry is provided:
    #       a- SPHERE(radius, facets)
    #       b- SPHERE(radius, facets, scalex, scaley, scalez)
    #       b- CUBE(sizex, sizey, sizez)
    #     RAND=factor: Defines a random factor factor 0 means that the particles are not deposited randomly
    #     ELLYPSE: defines the volume as an ellypse (default)
    #     RECTANGLE: defines the volume as a rectangle
    #     PROJECT: project the particles to the surface (default) (for welding, painting or scanning)
    #     NO_PROJECT: does not project the particles to the surface (for example, for 3D printing)
    #
    # volume (optional): Matrix of parameters defining the volume of the spray gun
    # geometry (optional): Matrix of vertices defining the triangles.

    if spray_id < 0:
        tool = 0  # auto detect active tool
        obj = 0  # auto detect object in active reference frame
        if Tool_Name is not None:
            tool = RDK.Item(Tool_Name, ITEM_TYPE_TOOL)

        if Object_Name is not None:
            obj = RDK.Item(Object_Name, ITEM_TYPE_OBJECT)
        # We can specify a given tool object and/or object
        #robot = RDK.Item("ABB IRB 2600-12/1.85", ITEM_TYPE_ROBOT)
        #tools = robot.Childs()
        #if len(tools) > 0:
        #    tool = tools[0]
        #obj = RDK.Item('object', ITEM_TYPE_OBJECT)

        # Create volume parameters
        options_command = "PROJECT PARTICLE=SPHERE(2,8,1,1,1) STEP=1x0 RAND=0 COLOR=" + COLOR

        spray_id = RDK.Spray_Add(tool, obj, options_command)

    # Remember the ID of the spray gun for later
    if Tool_Name is not None:
        RDK.setParam(Tool_Name, spray_id)

    # Apply the state to activate the trace
    RDK.Spray_SetState(SPRAY_ON, spray_id)

--- Python program ResetSoldar ---
# Type help("robodk.robolink") or help("robodk.robomath") for more information
# Press F5 to run the script
# Documentation: https://robodk.com/doc/en/RoboDK-API.html
# Reference:     https://robodk.com/doc/en/PythonAPI/robodk.html
# Note: It is not required to keep a copy of this file, your Python script is saved with your RDK project

# You can also use the new version of the API:
from robodk import robolink    # RoboDK API
from robodk import robomath    # Robot toolbox
RDK = robolink.Robolink()

RDK.Spray_Clear()

RDK.setParam('serigrafia', 0)
RDK.setParam('serigrafia1', 0)

--- Python program ConexionBasedeDatos ---
import psycopg
import random
import uuid


def conectar():
    conn = psycopg.connect(
        dbname="palillo",
        user="postgres",
        password="postgres",
        host="127.0.0.1",
        port="5432"
    )
    conn.execute("SET search_path TO produccion_palillos;")
    return conn


def crear_proceso_y_palillo():
    conn = conectar()
    cur = conn.cursor()

    # ==========================
    # 1. CREAR PROCESO
    # ==========================
    codigo_proceso = f"PR{uuid.uuid4().hex[:8]}"
    estado = random.choice(["en_curso", "finalizado", "error"])

    sql_proceso = """
    INSERT INTO produccion (cod_proceso, fecha_inicio, fecha_fin, estado)
    VALUES (%s, %s, %s, %s)
    """

    cur.execute(sql_proceso, (
        codigo_proceso,
        "2024-01-01",
        "2024-01-02",
        estado
    ))

    # ==========================
    # 2. CREAR PALILLO ASOCIADO
    # ==========================
    codigo_palillo = f"PL{uuid.uuid4().hex[:8]}"

    sql_palillo = """
    INSERT INTO palillo (codigo, forma, material_madera, grabado, cod_proceso)
    VALUES (%s, %s, %s, %s, %s)
    """

    cur.execute(sql_palillo, (
        codigo_palillo,
        random.choice(["alargado", "ovalado", "pequeño"]),
        random.choice(["roble", "pino", "cerezo", "reciclado"]),
        "estandar",
        codigo_proceso
    ))

    conn.commit()

    cur.close()
    conn.close()

    print(f"✔ Proceso creado: {codigo_proceso}")
    print(f"✔ Palillo creado: {codigo_palillo}")

--- Python program MqttListener ---
import paho.mqtt.client as mqtt
import RobotController as rc
from robodk import robolink
from robodk import robomath


RDK = robolink.Robolink()

broker="broker.emqx.io"
port=1883
base_topic_input="giirob/pr2/devices/input"
base_topic_output="giirob/pr2/devices/output"
station_input_topic_led=base_topic_input + "/led"
station_input_topic_led_2=base_topic_input + "/led2"
station_input_topic_lcd=base_topic_input + "/lcd"
station_output_topic=base_topic_output

def on_message(mqttc, obj, msg):
 payload = msg.payload.decode('utf-8')
 topic = msg.topic
 qos = msg.qos
 rc.handle_message(mqttc, topic, payload)

mqttc = mqtt.Client(mqtt.CallbackAPIVersion.VERSION2)
mqttc.on_message = on_message

def conectar_mqtt():
    mqttc.connect(broker, port, 60)
    mqttc.subscribe(station_output_topic, 0)
    print(f"INICIO DE LA ESTACIÓN")

def iniciar_loop_mqtt():
    mqttc.loop_start()

def encender_led():
    mqttc.publish(station_input_topic_led, "ENCENDER_LED")

def apagar_led():
    mqttc.publish(station_input_topic_led, "APAGAR_LED")

def encender_led_2():
    mqttc.publish(station_input_topic_led_2, "ENCENDER_LED")

def apagar_led_2():
    mqttc.publish(station_input_topic_led_2, "APAGAR_LED")

def publicar_lcd(mensaje):
    mqttc.publish(station_input_topic_lcd, mensaje)

--- Python program RobotController ---
from robodk import robolink # RoboDK API
from robodk import robomath # Robot toolbox
import MqttListener as mqtt_listener
RDK = robolink.Robolink()

def handle_message(mqttc, topic, payload):
    if topic == "giirob/pr2/devices/output":
        print(f"Payload recibido: {payload}")
        if payload == "PARAR":
            print ("Iniciando parada de emergencia...")
            RDK.setParam("stop", 1)   # Detiene la estación técnica

        elif payload == "INICIAR":
            print ("Reanudando operaciones...")
            RDK.setParam("stop", 0)   # Reanuda la estación técnica

        elif payload == "VACIO":
            print("Contenedor de palillos vacío")
            mqtt_listener.publicar_lcd("Contenedor vacio")

        elif payload == "LLENO":
            print("Contenedor de palillos lleno")
            mqtt_listener.publicar_lcd("Contenedor lleno")

        elif payload == "POCA_LUZ":
            print("Aumentar la iluminación")
            mqtt_listener.publicar_lcd("Aumentar luz")

        elif payload == "MUCHA_LUZ":
            print("Disminuir la iluminación")
            mqtt_listener.publicar_lcd("Disminuir luz")

        else:
            print ("Comando no reconocido.")
            mqtt_listener.publicar_lcd("Incorrect.")

--- Python program MainConveyor ---
from robodk import robolink
from robodk.robomath import transl, rotz
import time

RDK = robolink.Robolink()

FRAME = RDK.Item('MainConveyorRef', robolink.ITEM_TYPE_FRAME)

rack_base = RDK.Item('AssemblyRack', robolink.ITEM_TYPE_OBJECT)

STEP_GROUP = -970

MAX_BANDEJAS = 4

RDK.setParam('cinta_central', 0)

def esperar_stop():
    while int(RDK.getParam("stop") or 0) == 1:
        time.sleep(0.1)


def move_cinta_central(step=STEP_GROUP):

    esperar_stop()

    mechanism = RDK.Item('MainConveyor', robolink.ITEM_TYPE_ROBOT)

    if mechanism.Valid():
        j = mechanism.Joints()
        current = j[0, 0]
        mechanism.setJoints([current + float(step)])


def borrar_bandeja(group_id):

    esperar_stop()

    nombres = [
        f"bandeja_{group_id}_rack",
    ]

    for nombre in nombres:
        obj = RDK.Item(nombre)
        if obj.Valid():
            print("Eliminando:", nombre)
            obj.Delete()


def crear_bandeja(group_id, conveyor_position):

    esperar_stop()


    rack_base.Copy()
    rack = RDK.Paste()

    if rack.Valid():
        rack.setParent(FRAME)
        rack.setPose(transl(0, (-conveyor_position), 0))
        rack.setName(f"bandeja_{group_id}_rack")
    else:
        print("ERROR: No se pudo crear AssemblyRack")
        return False

    return True


def inicializar_bandejas():
    groups_on_belt = int(RDK.getParam('main_groups_on_belt') or 0)

    while groups_on_belt < MAX_BANDEJAS:
        esperar_stop()

        avanzar_y_crear_bandeja()
        groups_on_belt = int(RDK.getParam('main_groups_on_belt') or 0)

def avanzar_y_crear_bandeja():
    esperar_stop()

    conveyor_position = float(RDK.getParam('main_conv_pos') or 0)
    group_id = int(RDK.getParam('main_group_id') or 0)
    groups_on_belt = int(RDK.getParam('main_groups_on_belt') or 0)
    first_group_id = int(RDK.getParam('main_first_group_id') or 0)

    RDK.Render(False)

    ok = crear_bandeja(group_id, conveyor_position)

    if not ok:
        RDK.Render(True)
        return False

    conveyor_position -= STEP_GROUP
    RDK.setParam('main_conv_pos', conveyor_position)

    RDK.Render(True)

    RDK.setParam('cinta_central', 1)

    try:
        esperar_stop()
        move_cinta_central()
        time.sleep(0.5)
    finally:
        RDK.setParam('cinta_central', 0)

    group_id += 1
    groups_on_belt +=1

    RDK.setParam('main_group_id', group_id)
    RDK.setParam('main_groups_on_belt', groups_on_belt)
    RDK.setParam('main_first_group_id', first_group_id)

    RDK.Update()

    return True

--- Python program ResetMainConveyor ---
from robodk import robolink
import re

RDK = robolink.Robolink()

# -------------------------
# RESET PARÁMETROS
# -------------------------
RDK.setParam('main_conv_pos', 0)
RDK.setParam('main_group_id', 0)
RDK.setParam('main_groups_on_belt', 0)
RDK.setParam('main_first_group_id', 0)
RDK.setParam('cinta_central', 0)
RDK.setParam('correct_group_id', 0)
RDK.setParam('correct_groups_on_belt', 0)
RDK.setParam('correct_first_group_id', 0)

# -------------------------
# BUSCAR NOMBRES A ELIMINAR
# -------------------------
nombres_borrar = []

for item in RDK.ItemList():

    try:
        name = item.Name()
    except:
        continue

    if not name:
        continue

    if re.match(r"^bandeja_\d+_rack$", name) or re.match(r"^bandeja_\d+_plantilla$", name):
        nombres_borrar.append(name)

# -------------------------
# ELIMINAR OBJETOS
# -------------------------
for name in nombres_borrar:

    obj = RDK.Item(name)

    if obj.Valid():
        print("Eliminando:", name)
        obj.Delete()

# -------------------------
# DEVOLVER CINTA A ORIGEN
# -------------------------
mechanism = RDK.Item('MainConveyor', robolink.ITEM_TYPE_ROBOT)

if mechanism.Valid():
    joints = mechanism.Joints()
    joints[0, 0] = 0
    mechanism.setJoints(joints)

print("RESET CINTA CENTRAL COMPLETADO")

--- Python program ResetGeneral ---
from robodk import robolink

RDK = robolink.Robolink()

print("RESET GENERAL")

RDK.setParam('salir', 0)
RDK.setParam('stop', 0)
RDK.RunProgram("ResetDelta", True)
RDK.RunProgram("ResetStickConveyor", True)
RDK.RunProgram("ResetStickConveyorDeleteMove", True)
RDK.RunProgram("ResetMainConveyor", True)
RDK.RunProgram("ResetSoldar", True)
RDK.RunProgram("ResetPalillo")

print("RESET COMPLETADO")

--- Python program PararProgramas ---
from robodk import robolink

RDK = robolink.Robolink()

RDK.setParam("salir", 1)

--- Python program StopBoton ---
from robodk import robolink
import time

RDK = robolink.Robolink()

boton = RDK.Item('BotonStop')

if not boton.Valid():
    raise Exception("No existe BotonStop")

while int(RDK.getParam("salir") or 0) == 0:

    seleccion = RDK.Selection()

    if boton in seleccion:

        estado_actual = int(RDK.getParam('stop') or 0)

        if estado_actual == 0:
            RDK.setParam("stop", 1)
            print("STOP ACTIVADO")
        else:
            RDK.setParam("stop", 0)
            print("STOP DESACTIVADO")

        # Deseleccionar para que no se repita en bucle
        RDK.setSelection([])

    time.sleep(0.1)

--- Python program ProgramaPrincipal ---
from robodk import robolink
import time

RDK = robolink.Robolink()

print("CINTA ENTRADA")
RDK.RunProgram("StickConveyorMove")

# ESPERAR SOLO AL INICIO
while int(RDK.getParam("salir") or 0) == 0:

    groups_created = int(RDK.getParam("groups_created") or 0)

    print("Esperando grupos iniciales:", groups_created)

    if groups_created >= 5:
        break

    time.sleep(0.2)

print("CINTA SALIDA")
RDK.RunProgram("StickConveyorDeleteMove")

time.sleep(2)

print("SERIGRAFIA LASER")
RDK.RunProgram("SerigrafiaUR3e2")

time.sleep(1)

print("SERIGRAFIA LASER 1")
RDK.RunProgram("SerigrafiaUR3e1")

time.sleep(1)

print("BOTON STOP")
RDK.RunProgram("StopBoton")

time.sleep(2)

print("DELTA")
RDK.RunProgram("Delta")

print("SISTEMA INICIADO")
